FUNCTION_BLOCK AX_OR_8 (* FB to calculate boolean OR *)
  (* Standard: 61499-2; Description: Copyright (c) 2024 HR Agrartechnik GmbH This program and the accompanying materials are made available under the terms of the Eclipse Public License 2.0 which is available at https://www.eclipse.org/legal/epl-2.0/ SPDX-License-Identifier: EPL-2.0 *)
  (* Version 1.0, 2024-10-23, Franz Höpfinger, HR Agrartechnik GmbH *)
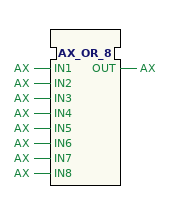
  SOCKETS
    IN1 : AX; (* OR input 1 *)
    IN2 : AX; (* OR input 2 *)
    IN3 : AX; (* OR input 3 *)
    IN4 : AX; (* OR input 4 *)
    IN5 : AX; (* OR input 5 *)
    IN6 : AX; (* OR input 6 *)
    IN7 : AX; (* OR input 7 *)
    IN8 : AX; (* OR input 8 *)
  END_SOCKETS
  PLUGS
    OUT : AX; (* OR result *)
  END_PLUGS
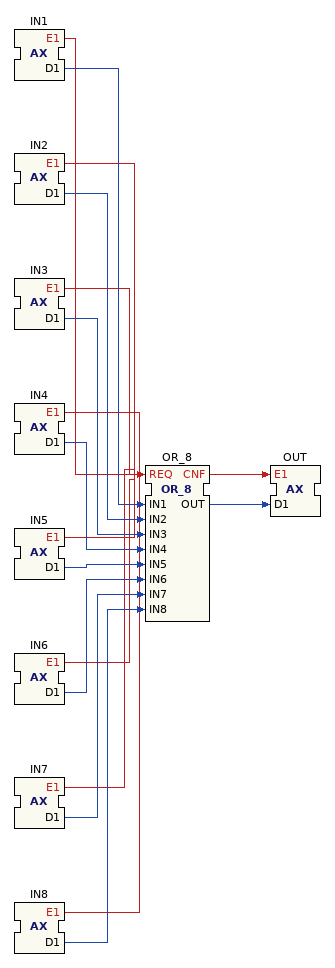
  FBS
    OR_8 : OR_8;
  END_FBS
  EVENT_CONNECTIONS
    IN1.E1 TO OR_8.REQ;
    IN2.E1 TO OR_8.REQ;
    OR_8.CNF TO OUT.E1;
    IN3.E1 TO OR_8.REQ;
    IN4.E1 TO OR_8.REQ;
    IN5.E1 TO OR_8.REQ;
    IN6.E1 TO OR_8.REQ;
    IN7.E1 TO OR_8.REQ;
    IN8.E1 TO OR_8.REQ;
  END_CONNECTIONS
  DATA_CONNECTIONS
    IN1.D1 TO OR_8.IN1;
    IN2.D1 TO OR_8.IN2;
    OR_8.OUT TO OUT.D1;
    IN3.D1 TO OR_8.IN3;
    IN4.D1 TO OR_8.IN4;
    IN5.D1 TO OR_8.IN5;
    IN6.D1 TO OR_8.IN6;
    IN7.D1 TO OR_8.IN7;
    IN8.D1 TO OR_8.IN8;
  END_CONNECTIONS
END_FUNCTION_BLOCK
